(* PLC project Unnamed, Unknown Unnamed 1 *)
(* stored: creationDateTime 2026-06-10T17:03:42, modificationDateTime 2026-06-10T17:03:42 *)

PROGRAM main
  VAR
    Q_READY AT %QX0.0 : BOOL := False;
    Q_REQUEST AT %QX0.1 : BOOL := False;
    Q_PASS_ALLOWED AT %QX0.2 : BOOL := False;
    Q_EMERGENCY AT %QX0.3 : BOOL := False;
    CMD_ROBOT_REQUEST AT %QX1.0 : BOOL := False;
    CMD_HMI_ALLOW AT %QX1.1 : BOOL := False;
    CMD_ROBOT_PASSED AT %QX1.2 : BOOL := False;
    CMD_EMERGENCY AT %QX1.3 : BOOL := False;
    CMD_RESET AT %QX1.4 : BOOL := False;
    STATUS_READY AT %QX0.4 : BOOL := False;
    STATUS_REQUEST AT %QX0.5 : BOOL := False;
    STATUS_PASS_ALLOWED AT %QX0.6 : BOOL := False;
    STATUS_EMERGENCY AT %QX0.7 : BOOL := False;
  END_VAR
  VAR
    STATUS_BARRIER_OPEN : BOOL := False;
    STATUS_PASS_PERMISSION : BOOL := False;
    M_READY : BOOL := True;
    M_REQUEST : BOOL := False;
    M_PASS_ALLOWED : BOOL := False;
    M_EMERGENCY : BOOL := False;
    PWM_CONTROLLER0 : PWM_CONTROLLER;
    SERVO_CHANNEL : SINT := 13;
    SERVO_FREQ : REAL := 50.0;
    SERVO_DUTY_CLOSED : REAL := 5.0;
    SERVO_DUTY_OPEN : REAL := 7.5;
    PWM_CLOSE_OK : BOOL := False;
    PWM_OPEN_OK : BOOL := False;
  END_VAR

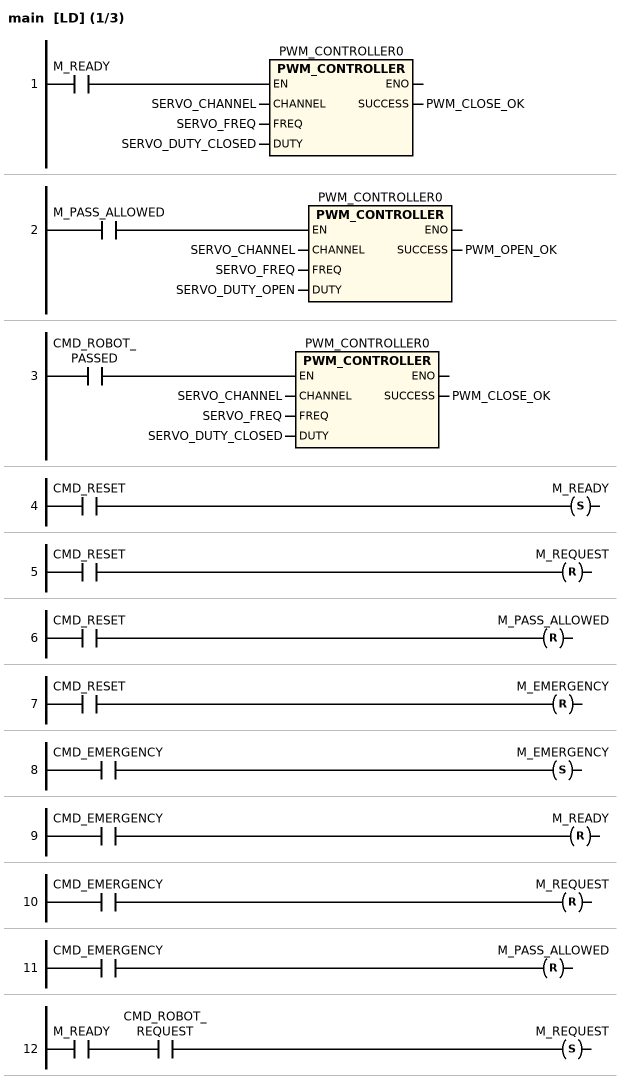
(* LD diagram, written out as Structured Text *)
IF CMD_RESET THEN M_READY := TRUE; END_IF;
IF CMD_RESET THEN M_REQUEST := FALSE; END_IF;
IF CMD_RESET THEN M_PASS_ALLOWED := FALSE; END_IF;
IF CMD_RESET THEN M_EMERGENCY := FALSE; END_IF;
IF CMD_EMERGENCY THEN M_EMERGENCY := TRUE; END_IF;
IF CMD_EMERGENCY THEN M_READY := FALSE; END_IF;
IF CMD_EMERGENCY THEN M_REQUEST := FALSE; END_IF;
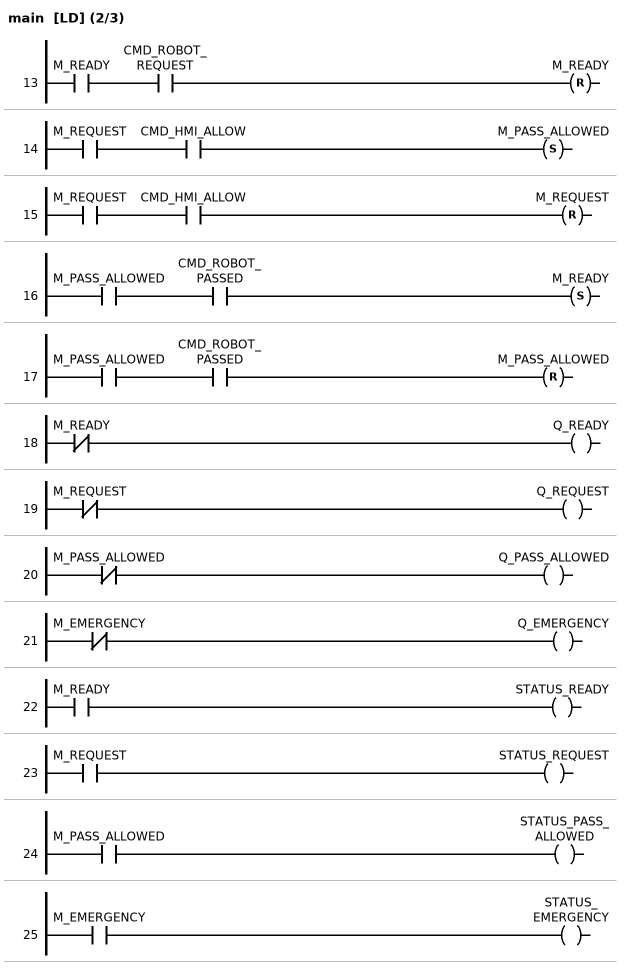
IF CMD_EMERGENCY THEN M_PASS_ALLOWED := FALSE; END_IF;
IF M_READY AND CMD_ROBOT_REQUEST THEN M_REQUEST := TRUE; END_IF;
IF M_READY AND CMD_ROBOT_REQUEST THEN M_READY := FALSE; END_IF;
IF M_REQUEST AND CMD_HMI_ALLOW THEN M_PASS_ALLOWED := TRUE; END_IF;
IF M_REQUEST AND CMD_HMI_ALLOW THEN M_REQUEST := FALSE; END_IF;
IF M_PASS_ALLOWED AND CMD_ROBOT_PASSED THEN M_READY := TRUE; END_IF;
IF M_PASS_ALLOWED AND CMD_ROBOT_PASSED THEN M_PASS_ALLOWED := FALSE; END_IF;
Q_READY := NOT M_READY;
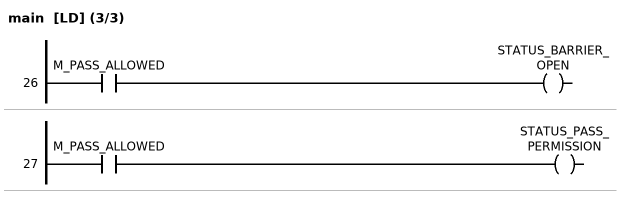
Q_REQUEST := NOT M_REQUEST;
Q_PASS_ALLOWED := NOT M_PASS_ALLOWED;
Q_EMERGENCY := NOT M_EMERGENCY;
STATUS_READY := M_READY;
STATUS_REQUEST := M_REQUEST;
STATUS_PASS_ALLOWED := M_PASS_ALLOWED;
STATUS_EMERGENCY := M_EMERGENCY;
STATUS_BARRIER_OPEN := M_PASS_ALLOWED;
STATUS_PASS_PERMISSION := M_PASS_ALLOWED;
PWM_CONTROLLER0(EN := M_READY, CHANNEL := SERVO_CHANNEL, FREQ := SERVO_FREQ, DUTY := SERVO_DUTY_CLOSED);
IF PWM_CONTROLLER0.ENO THEN PWM_CLOSE_OK := PWM_CONTROLLER0.SUCCESS; END_IF;
PWM_CONTROLLER0(EN := M_PASS_ALLOWED, CHANNEL := SERVO_CHANNEL, FREQ := SERVO_FREQ, DUTY := SERVO_DUTY_OPEN);
IF PWM_CONTROLLER0.ENO THEN PWM_OPEN_OK := PWM_CONTROLLER0.SUCCESS; END_IF;
PWM_CONTROLLER0(EN := CMD_ROBOT_PASSED, CHANNEL := SERVO_CHANNEL, FREQ := SERVO_FREQ, DUTY := SERVO_DUTY_CLOSED);
IF PWM_CONTROLLER0.ENO THEN PWM_CLOSE_OK := PWM_CONTROLLER0.SUCCESS; END_IF;
END_PROGRAM

CONFIGURATION Config0
  RESOURCE Res0 ON PLC
    TASK task0(INTERVAL := T#20ms, PRIORITY := 1);
    PROGRAM instance0 WITH task0 : main;
  END_RESOURCE
END_CONFIGURATION
